FUNCTION_BLOCK Controller

VAR_OUTPUT
	
END_VAR

VAR	
	// 輸入指令，顯示狀態、位置、角度
	command : E_6Axis_Command;	
	state : ST_6Axis_State;
	constructState : UINT;
	touchingState : UINT;
	takeState : UINT;
	JointDegNow : ARRAY [AXIS_MIN_IDX..AXIS_MAX_IDX] OF LREAL;
	PositionNow : ARRAY [AXIS_MIN_IDX..AXIS_MAX_IDX] OF LREAL;
	hasFromCAM : BOOL;
	//StartPosition_Now : ARRAY [AXIS_MIN_IDX..AXIS_MAX_IDX] OF LREAL; // for linear move used
	
	// 開發者使用
	HomePoint : ARRAY [AXIS_MIN_IDX..AXIS_MAX_IDX] OF LREAL := [565, 0, 834, 0, 0, 0];
	HomeJoint : ARRAY [AXIS_MIN_IDX..AXIS_MAX_IDX] OF LREAL := [0, 0, 0, 0, 0, 0]; // for joints space	

	//BufferMot : Motion_Command_Input; // 
	InitalPOS : ARRAY [AXIS_MIN_IDX..AXIS_MAX_IDX] OF LREAL := InitalPOS;
	ActExecute : BOOL := FALSE;
	ExecutePMD : BOOL := FALSE;
	ExecuteCAL : BOOL := FALSE; // 執行一次性計算
 	DIR : LREAL := 0; // XYZ_Direcation XYZ軸方向 = {1:x, 2:y, 3:z, 4:xy, 5:-(xy)}
	PMD : LREAL := 0; // Path_Motion_Displace 路徑移動距離
	TouchDetection : BOOL;
	ZeroArray : ARRAY [AXIS_MIN_IDX..AXIS_MAX_IDX] OF LREAL := [0, 0, 0, 0, 0, 0]; 
	TargetPOS : ARRAY [AXIS_MIN_IDX..AXIS_MAX_IDX] OF LREAL := [650, -150, 500, -42, 0, 45];
	POS_STORAGE : Buffer;

	// 索引
	idx : USINT(AXIS_MIN_IDX..AXIS_MAX_IDX);
	movableBlock_idx : INT;
	i, j : USINT(AXIS_MIN_IDX..AXIS_MAX_IDX);
	z : INT;
	n : ARRAY [1..6] OF LREAL := AutoMotionData.CAMStore[1][0] ;
	usingMotion : INT;
	row, col : INT;
	//ok
	//p : ARRAY [1..2] OF LREAL := AutoMotionData.CAMStore;
	//L : ARRAY [AXIS_MIN_IDX..AXIS_MAX_IDX] OF LREAL ;
	h : INT;
	

	// 基本需要的函式
	Axis : ARRAY[AXIS_MIN_IDX..AXIS_MAX_IDX] OF AXIS_REF;
	Power : ARRAY [AXIS_MIN_IDX..AXIS_MAX_IDX] OF MC_Power;
	Stop : ARRAY [AXIS_MIN_IDX..AXIS_MAX_IDX] OF MC_Stop; //delete
	Halt : ARRAY [AXIS_MIN_IDX..AXIS_MAX_IDX] OF MC_Halt; 
	Reset : ARRAY [AXIS_MIN_IDX..AXIS_MAX_IDX] OF MC_Reset;
	
	// 自訂義函式
	KM : Kinematics;
	MF : MathFunc;
	
	// 移動用函式
	AbsMove : ARRAY [AXIS_MIN_IDX..AXIS_MAX_IDX] OF MC_MoveAbsolute;
	ExtSwitchEn : ARRAY [AXIS_MIN_IDX..AXIS_MAX_IDX] OF MC_ExtSetPointGenEnable;
	ExtSwitchDis : ARRAY [AXIS_MIN_IDX..AXIS_MAX_IDX] OF MC_ExtSetPointGenDisable;
	LinearMove : MC_Linear; 

	// For Curve                         A1  A2  A3  A4  A5  A6
	StartVEL : ARRAY [1..6] OF LREAL := [  0,  0,  0,  0,  0,  0];
	StartACC : ARRAY [1..6] OF LREAL := [  0,  0,  0,  0,  0,  0];
	FinalVEL : ARRAY [1..6] OF LREAL := [  0,  0,  0,  0,  0,  0];
	FinalACC : ARRAY [1..6] OF LREAL := [  0,  0,  0,  0,  0,  0];

	E_Command: INT;
	No_Command: INT;
	PT: TIME;
END_VAR

readAxis();
SetStartPosition();

CASE command OF
	E_6Axis_Command.NO_COMMAND:
		FOR idx := AXIS_MIN_IDX TO AXIS_MAX_IDX DO
			AbsMove[idx].Execute := FALSE;
		END_FOR
		isHalt := FALSE;
		ExecutePMD := FALSE;
		constructState := 0;
		ActExecute := FALSE;
		
	E_6Axis_Command.POWER_ON:
		FOR idx := AXIS_MIN_IDX TO AXIS_MAX_IDX DO
			Power[idx].Enable := TRUE;
		END_FOR
		IF state.powerOn THEN
			command := E_6Axis_Command.HOMING;
		END_IF
	
	E_6Axis_Command.HALT:
		FOR idx := AXIS_MIN_IDX TO AXIS_MAX_IDX DO
			Halt[idx].Execute := TRUE;
		END_FOR
		IF NOT state.moving THEN
			FOR idx := AXIS_MIN_IDX TO AXIS_MAX_IDX DO
				Halt[idx].Execute := FALSE;
			END_FOR
		END_IF
		command := E_6axis_Command.NO_COMMAND;
	
	E_6Axis_Command.RESET:
		FOR idx := AXIS_MIN_IDX TO AXIS_MAX_IDX DO
			Reset[idx].Execute := TRUE;
			IF Reset[idx].Done THEN
				Reset[idx].Execute := FALSE;
			END_IF
		END_FOR
		command := E_6axis_Command.NO_COMMAND;

	// SetMotion(路徑模式，起點，終點，FALSE);		
	E_6Axis_Command.HOMING:
		ActExecute := TRUE;
		SetMotion(0, InitalPOS, HomeJoint, FALSE, TRUE);
		IF NOT ActExecute THEN
			command := E_6axis_Command.NO_COMMAND;
		END_IF

	E_6Axis_Command.M_PTP:
		ActExecute := TRUE;
		SetMotion(0, InitalPOS, TargetPOS, FALSE, FALSE);
		IF NOT ActExecute THEN
			command := E_6axis_Command.NO_COMMAND;
		END_IF
		
	E_6Axis_Command.M_DIRE_X:
		IF NOT ExecutePMD THEN
			MF.VectorMotionPOS(POS := TargetPOS, DIR, PMD);
			ExecutePMD := TRUE;
		END_IF
		ActExecute := TRUE;
		SetMotion(1, InitalPOS, TargetPOS, FALSE, FALSE);
		IF NOT ActExecute THEN
			command := E_6axis_Command.NO_COMMAND;
		END_IF
		
	E_6Axis_Command.M_DIRE_Y:
		IF NOT ExecutePMD THEN
			MF.VectorMotionPOS(POS := TargetPOS, DIR, PMD);
			ExecutePMD := TRUE;
		END_IF
		ActExecute := TRUE;
		SetMotion(1, InitalPOS, TargetPOS, FALSE, FALSE);
		IF NOT ActExecute THEN
			command := E_6axis_Command.NO_COMMAND;
		END_IF
	
	E_6Axis_Command.M_DIRE_XY:
		IF NOT ExecutePMD THEN
			MF.VectorMotionPOS(POS := TargetPOS, DIR, PMD);
			ExecutePMD := TRUE;
		END_IF
		ActExecute := TRUE;
		SetMotion(1, InitalPOS, TargetPOS, FALSE, FALSE);
		IF NOT ActExecute THEN
			command := E_6axis_Command.NO_COMMAND;
		END_IF
		
	E_6Axis_Command.M_DIRE_Z:
		IF NOT ExecutePMD THEN
			MF.VectorMotionPOS(POS := TargetPOS, DIR, PMD);
			ExecutePMD := TRUE;
		END_IF
		ActExecute := TRUE;
		SetMotion(1, InitalPOS, TargetPOS, FALSE, FALSE);
		IF NOT ActExecute THEN
			command := E_6axis_Command.NO_COMMAND;
		END_IF
		
	E_6Axis_Command.M_LINEAR:
		ActExecute := TRUE;
		SetMotion(1, InitalPOS, TargetPOS, FALSE, FALSE);
		IF NOT ActExecute THEN
			command := E_6axis_Command.NO_COMMAND;
		END_IF
		
	E_6Axis_Command.M_CURVE:
		ActExecute := TRUE;
		SetMotion(2, InitalPOS, TargetPOS, FALSE, FALSE);
		IF NOT ActExecute THEN
			command := E_6axis_Command.NO_COMMAND;
		END_IF
		
	E_6Axis_Command.TOUCHING://判斷式
		IF NOT ActExecute THEN
			CASE touchingState OF
				0: //要再加一個判斷式判斷是哪一個位置
					//z := z + 1;            // 疊疊樂右面與左面
					usingMotion := 2;
					
					IF z = 1 THEN
						TargetPOS[1]:= n[1];
						TargetPOS[2]:= n[2];
						TargetPOS[3]:= 500;
						TargetPOS[4]:= 0;
						TargetPOS[5]:= 90;
						TargetPOS[6]:= -45;
					ELSIF z = 2 THEN
						TargetPOS[1]:= n[1];
						TargetPOS[2]:= n[2];
						TargetPOS[3]:= 500;
						TargetPOS[4]:= 0;
						TargetPOS[5]:= 90;
						TargetPOS[6]:= -135;
					END_IF
					      // 移動模式
					//TargetPOS := AutoMotionData.CAMStore[n][z];  // n=0
					//n := n + 1;
					touchingState := touchingState + 1;
				1:
					usingMotion := 1;
					IF z = 1 THEN
						MF.VectorMotionPOS(POS := TargetPOS, 5, -25);
					ELSIF z = 2 THEN
						MF.VectorMotionPOS(POS := TargetPOS, 4, 25);
					END_IF
					//AutoMotionData.POStore[z][n] := TargetPOS;
					//n := n + 1;
					touchingState := touchingState + 1;
				2: 
					usingMotion := 1;
					IF z = 1 THEN
						MF.VectorMotionPOS(POS := TargetPOS, 3, -(500-n[3]));
					ELSIF z = 2 THEN
						MF.VectorMotionPOS(POS := TargetPOS, 3, -(500-n[3]));
					END_IF
					touchingState := touchingState + 1;
				3:
					PT := T#1S;
					input_dig[1] := TRUE;
					PT := T#1S;
					//加計時器
					input_dig[1] := FALSE;
				4:
					usingMotion := 1;
					IF z = 1 THEN
						MF.VectorMotionPOS(POS := TargetPOS, 3, (500-n[3]));
					ELSIF z = 2 THEN
						MF.VectorMotionPOS(POS := TargetPOS, 3, (500-n[3]));
					END_IF
					touchingState := touchingState + 1;
				
				5:
					command := E_6axis_Command.HOMING;
					touchingState := touchingState + 1;
				6:
					command := E_6axis_Command.TAKING;
			END_CASE			
		END_IF
	SetMotion(usingMotion, InitalPOS, TargetPOS, FALSE, FALSE);
	
	E_6Axis_Command.TAKING:
		IF NOT ActExecute THEN
			CASE takeState OF
				0:
					usingMotion := 1;
					input_dig[2] := FALSE;
					
					IF z = 1 THEN
						MF.VectorMotionPOS(POS := TargetPOS, 5, (n[1]+100));
						MF.VectorMotionPOS(POS := TargetPOS, 5, (n[2]+100));
						TargetPOS[3] := 500;
						TargetPOS[4] := 0;
						TargetPOS[5] := -90;
						TargetPOS[6] := 45;
					ELSIF z = 2 THEN
						MF.VectorMotionPOS(POS := TargetPOS, 4, (n[1]-100));
						MF.VectorMotionPOS(POS := TargetPOS, 4, (n[2]-100));
						TargetPOS[3] := 500;
						TargetPOS[4] := 0;
						TargetPOS[5] := -90;
						TargetPOS[6] := -135;
						
					END_IF
					touchingState := touchingState + 1;	
				1:
					usingMotion := 1;
					IF z = 1 THEN
						MF.VectorMotionPOS(POS := TargetPOS, 3, -(500-n[3]));
					ELSIF z = 2 THEN
						MF.VectorMotionPOS(POS := TargetPOS, 3, -(500-n[3]));
					END_IF
					//AutoMotionData.POStore[z][n] := hasFromCAM;
					//n := n + 1;
					touchingState := touchingState + 1;
				2:
					usingMotion := 1; 
					input_dig[2]:= TRUE ;
					PT := T#1S;
					touchingState := touchingState + 1;
				3:
					usingMotion := 1; 
					IF z = 1 THEN
						MF.VectorMotionPOS(POS := TargetPOS, 5, 30);
					ELSIF z = 2 THEN
						MF.VectorMotionPOS(POS := TargetPOS, 4, -30);
					END_IF
					touchingState := touchingState + 1;
				4:
					usingMotion := 1;
					
					MF.VectorMotionPOS(POS := TargetPOS, 3, (AutoMotionData.Heightstore[1]-n[3]+2));
					touchingState := touchingState + 1;
				5:
				   IF z = 1 THEN
						MF.VectorMotionPOS(POS := TargetPOS, 5, -60);
					ELSIF z = 2 THEN
						MF.VectorMotionPOS(POS := TargetPOS, 4, 60);
					END_IF
					PT := T#1S;
					input_dig[2]:= FALSE ;
					touchingState := touchingState + 1;
				6:
					command := E_6axis_Command.HOMING;
					
			END_CASE
		END_IF
		SetMotion(usingMotion, InitalPOS, TargetPOS, FALSE, FALSE);
		ActExecute := TRUE;
				
				
//	E_6Axis_Command.LOOKING:
//		SetMotion(0, InitalPOS, TargetPOS, FALSE);

END_CASE

Decider();
Update_AbsMove_Motion();
Update_Custom_Motion();
ActPower();
ActReset();
ActStop();

//	E_6Axis_Command.CONSTRUCT:
//		IF NOT ActExecute THEN
//			CASE constructState OF
//				0:
//					z := z + 1;            // 疊疊樂右面與左面
//					usingMotion := 2;      // 移動模式
//					TargetPOS := AutoMotionData.POStore[z][n];  // n=0
//					n := n + 1;
//					constructState := constructState + 1;
//				1:
//					usingMotion := 1;
//					IF z = 1 THEN
//						MF.VectorMotionPOS(POS := TargetPOS, 4, 90);
//					ELSIF z = 2 THEN
//						MF.VectorMotionPOS(POS := TargetPOS, 5, 90);
//					END_IF
//					AutoMotionData.POStore[z][n] := TargetPOS;
//					n := n + 1;
//					constructState := constructState + 1;
//				2:
//					usingMotion := 1;
//					IF z = 1 THEN
//						MF.VectorMotionPOS(POS := TargetPOS, 3, -95);
//					ELSIF z = 2 THEN
//						MF.VectorMotionPOS(POS := TargetPOS, 3, -110);
//					END_IF					
//					AutoMotionData.POStore[z][n] := TargetPOS;
//					n := n + 1;
//					constructState := constructState + 1;
//				3:
//					usingMotion := 1;
//					TouchDetection := TRUE;
//					ExecuteCAL := FALSE;
//					IF z = 1 THEN
//						MF.VectorMotionPOS(POS := TargetPOS, 4, -40);
//					ELSIF z = 2 THEN
//						MF.VectorMotionPOS(POS := TargetPOS, 5, -40);
//					END_IF	
//					AutoMotionData.POStore[z][n] := TargetPOS;
//					n := n + 1;
//					movableBlock_idx := movableBlock_idx + 1;
//					constructState := constructState + 1;
//				4:
//					usingMotion := 1;
//					TouchDetection := FALSE;
//					row := row + 1;
//					IF z = 1 THEN
//						MF.VectorMotionPOS(POS := TargetPOS, 4, 40);
//					ELSIF z = 2 THEN
//						MF.VectorMotionPOS(POS := TargetPOS, 5, 40);
//					END_IF	
//					AutoMotionData.POStore[z][n] := TargetPOS;
//					n := n + 1; 
//					constructState := constructState + 1;
//					IF row = 3 THEN
//						row := 0;
//						constructState := 6;
//						col := col + 1;
//						IF col = 4 THEN
//							constructState := 8;
//						END_IF
//					END_IF
//				5:
//					usingMotion := 1;
//					IF z = 1 THEN
//						MF.VectorMotionPOS(POS := TargetPOS, 5, -25);
//					ELSIF z = 2 THEN
//						MF.VectorMotionPOS(POS := TargetPOS, 4, -25);
//					END_IF	
//					AutoMotionData.POStore[z][n] := TargetPOS;
//					n := n + 1;
//					constructState := 3;
//				6:
//					usingMotion := 1;
//					MF.VectorMotionPOS(POS := TargetPOS, 3, -30);
//					AutoMotionData.POStore[z][n] := TargetPOS;
//					n := n + 1;
//					constructState := constructState + 1;
//				7:
//					usingMotion := 1;
//					IF z = 1 THEN
//						MF.VectorMotionPOS(POS := TargetPOS, 5, 50);
//					ELSIF z = 2 THEN
//						MF.VectorMotionPOS(POS := TargetPOS, 4, 50);
//					END_IF	
//					AutoMotionData.POStore[z][n] := TargetPOS;
//					n := n + 1;
//					constructState := 3;
//				8:
//					usingMotion := 2;
//					TargetPOS := AutoMotionData.POStore[z][1];
//					constructState := 9;
//				9:
//					usingMotion := 2;
//					TargetPOS := HomePoint;
//					n := 0;
//					row := 0;
//					col := 0;
//					constructState := 0;
//					IF z = 2 THEN
//						constructState := 10;
//					END_IF
//				10:
//					command := E_6axis_Command.HOMING;
//					constructState := 11;
//			END_CASE
//		END_IF
//		ActExecute := TRUE;
//		IF TouchDetection THEN
//			IF input_dig[1] THEN
//				IF NOT ExecuteCAL THEN
//					AutoMotionData.MovableBlocks[movableBlock_idx] := ZeroArray;
//					movableBlock_idx := movableBlock_idx - 1;
//					ExecuteCAL := TRUE;
//				END_IF
//			ELSE
//				// 減2是為了擷取上一個座標
//				AutoMotionData.MovableBlocks[movableBlock_idx] := AutoMotionData.POStore[z][n-2];
//			END_IF
//		END_IF

//		IF NOT (constructState = 11) THEN
//			SetMotion(usingMotion, InitalPOS, TargetPOS, FALSE, FALSE);
//		ELSE
//			z := 0;
//		END_IF

ACTION ActHalt:
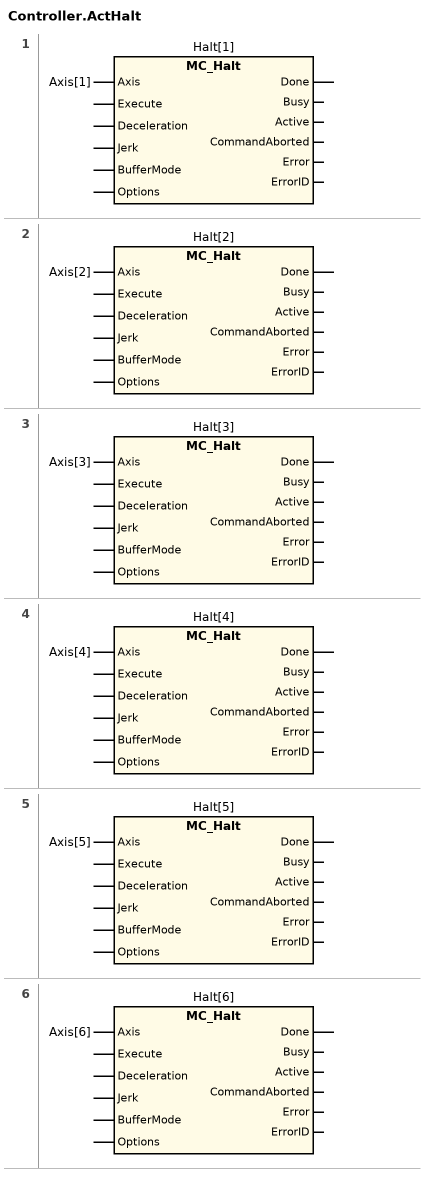
// NETWORK 1
Halt[1](Axis := Axis[1]); // MC_Halt

// NETWORK 2
Halt[2](Axis := Axis[2]); // MC_Halt

// NETWORK 3
Halt[3](Axis := Axis[3]); // MC_Halt

// NETWORK 4
Halt[4](Axis := Axis[4]); // MC_Halt

// NETWORK 5
Halt[5](Axis := Axis[5]); // MC_Halt

// NETWORK 6
Halt[6](Axis := Axis[6]); // MC_Halt
END_ACTION

ACTION ActPower:
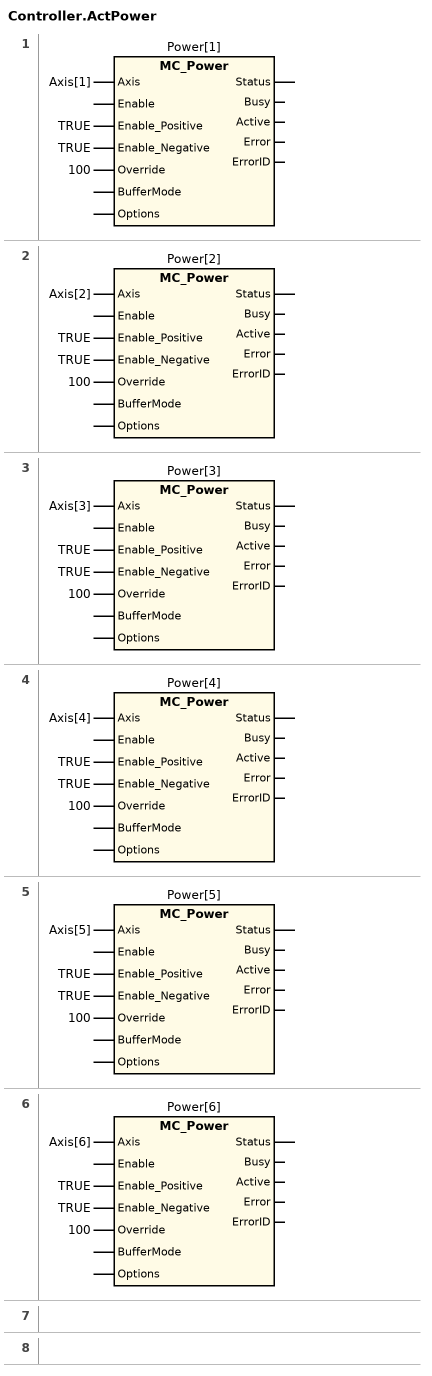
// NETWORK 1
Power[1](Axis := Axis[1], Enable_Positive := TRUE, Enable_Negative := TRUE, Override := 100); // MC_Power

// NETWORK 2
Power[2](Axis := Axis[2], Enable_Positive := TRUE, Enable_Negative := TRUE, Override := 100); // MC_Power

// NETWORK 3
Power[3](Axis := Axis[3], Enable_Positive := TRUE, Enable_Negative := TRUE, Override := 100); // MC_Power

// NETWORK 4
Power[4](Axis := Axis[4], Enable_Positive := TRUE, Enable_Negative := TRUE, Override := 100); // MC_Power

// NETWORK 5
Power[5](Axis := Axis[5], Enable_Positive := TRUE, Enable_Negative := TRUE, Override := 100); // MC_Power

// NETWORK 6
Power[6](Axis := Axis[6], Enable_Positive := TRUE, Enable_Negative := TRUE, Override := 100); // MC_Power

// NETWORK 7

// NETWORK 8
END_ACTION

ACTION ActReset:
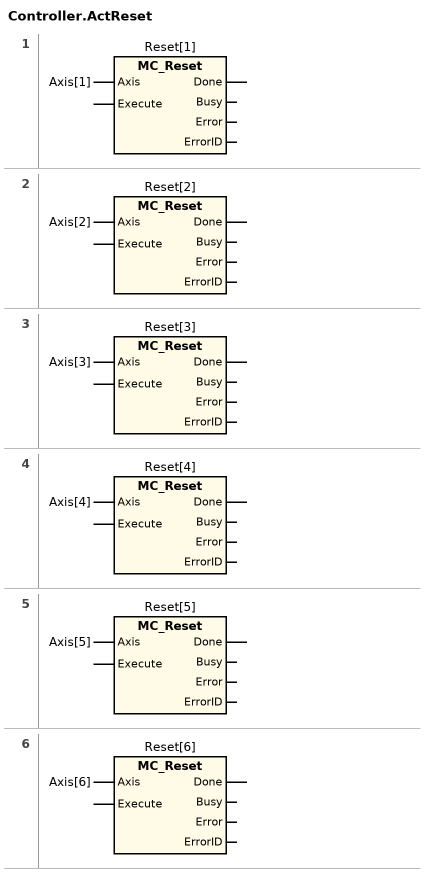
// NETWORK 1
Reset[1](Axis := Axis[1]); // MC_Reset

// NETWORK 2
Reset[2](Axis := Axis[2]); // MC_Reset

// NETWORK 3
Reset[3](Axis := Axis[3]); // MC_Reset

// NETWORK 4
Reset[4](Axis := Axis[4]); // MC_Reset

// NETWORK 5
Reset[5](Axis := Axis[5]); // MC_Reset

// NETWORK 6
Reset[6](Axis := Axis[6]); // MC_Reset
END_ACTION

ACTION ActStop:
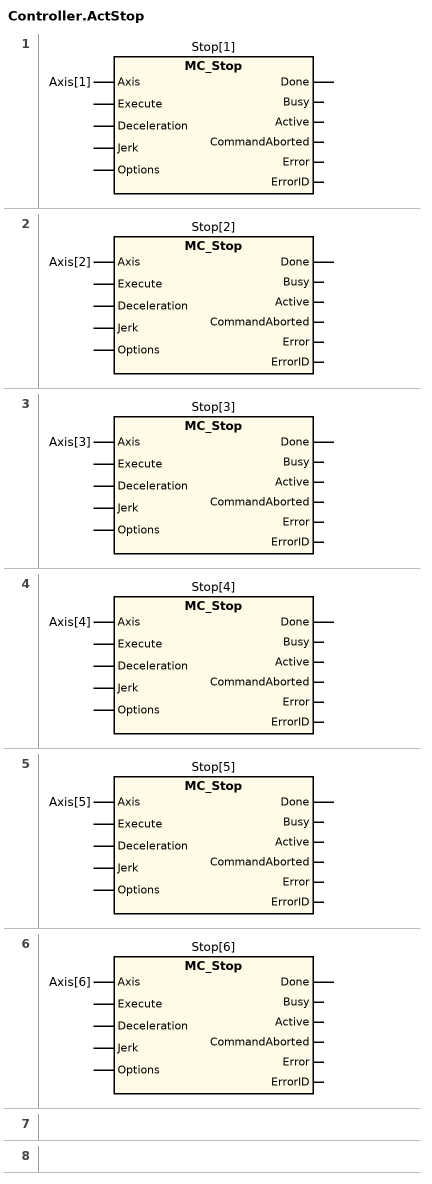
// NETWORK 1
Stop[1](Axis := Axis[1]); // MC_Stop

// NETWORK 2
Stop[2](Axis := Axis[2]); // MC_Stop

// NETWORK 3
Stop[3](Axis := Axis[3]); // MC_Stop

// NETWORK 4
Stop[4](Axis := Axis[4]); // MC_Stop

// NETWORK 5
Stop[5](Axis := Axis[5]); // MC_Stop

// NETWORK 6
Stop[6](Axis := Axis[6]); // MC_Stop

// NETWORK 7

// NETWORK 8
END_ACTION

ACTION Decider:
IF NOT state.moving AND AbsMove[1].Done AND AbsMove[2].Done AND AbsMove[3].Done AND AbsMove[4].Done  AND AbsMove[5].Done AND AbsMove[6].Done THEN
	command := E_6axis_Command.NO_COMMAND;	
END_IF

IF state.error THEN
	command := E_6Axis_Command.RESET;
END_IF

IF isHalt THEN
	command := E_6Axis_Command.HALT;
END_IF
END_ACTION

METHOD mode_Curve : BOOL

VAR_INPUT
	six_mat : ARRAY [1..6, 1..6] OF LREAL;
END_VAR

VAR_OUTPUT
	execute_fullTime : LREAL;
	coeffCopy : ARRAY [1..6, 1..6] OF LREAL;
END_VAR

VAR
	idx : DINT;
	i, j : INT;
	t : LREAL;
	temp : LREAL; // 導正係數用
	
	startAngles : ARRAY [1..6] OF LREAL;
	finalAngles : ARRAY [1..6] OF LREAL;
	pos01, pos02 : ARRAY [1..3] OF LREAL; //start and final point for calculate fulltime
	
	six_matCopy : ARRAY [1..6, 1..6] OF LREAL;
	TimeMatrix : ARRAY [1..6, 1..6] OF LREAL;
END_VAR
// Angles_mat
six_matCopy := six_mat;  // 含有角度 := 含有座標
FOR idx := 1 TO 6 DO 
	IF (idx < 3) THEN
		pos01[idx] := six_mat[idx, 1];
		pos02[idx] := six_mat[idx, 4];
	END_IF
	startAngles[idx] := six_mat[idx, 1];
	finalAngles[idx] := six_mat[idx, 4];
END_FOR
KM.Inverse(position := startAngles, degrees => startAngles);
KM.Inverse(position := finalAngles, degrees => finalAngles);
FOR idx := 1 TO 6 DO 
	six_matCopy[idx, 1] := startAngles[idx];
	six_matCopy[idx, 4] := finalAngles[idx];
END_FOR

MF.FindFullTime(pos01, pos02, 10, execute_fullTime => execute_fullTime);
t := execute_fullTime;
// Time_mat
FOR i := 1 TO 6 DO
    FOR j := 1 TO 6 DO
        CASE j OF
            1: 
                // 第一列固定為1、0、0、0、0、0
                TimeMatrix[i, j] := SEL(i = 1, 0, 1);
            2: 
                // 第二列固定為0、1、0、0、0、0
                TimeMatrix[i, j] := SEL(i = 2, 0, 1);
            3:
                // 第三列固定為0、0、2、0、0、0
                TimeMatrix[i, j] := SEL(i = 3, 0, 2);
            4:
                // 第四列公式：1 * EXPT(t, i)
                TimeMatrix[i, j] := EXPT(t, i-1);
            5:
                // 第五列公式：i * EXPT(t, i-1)
                TimeMatrix[i, j] := (i-1) * EXPT(t, i-2);
            6:
                // 第六列公式：(i * (i - 1)) * EXPT(t, i-2)
                TimeMatrix[i, j] := (i-1) * (i-2) * EXPT(t, i-3);
        END_CASE
    END_FOR
END_FOR

MF.GaussianElimination(base_mat := TimeMatrix, extend_mat := six_matCopy, temp_mat := coeffCopy, 6); //inverse 會搞壞原本的東西

FOR i := 1 TO 6 DO
	FOR j := 1 TO 3 DO
		temp := coeffCopy[i, j];
		coeffCopy[i, j] := coeffCopy[i, 7-j];
		coeffCopy[i, 7-j] := temp;
	END_FOR		
END_FOR
END_METHOD

METHOD mode_Linear : BOOL

VAR_INPUT
	six_pos : ARRAY [1..6, 1..6] OF LREAL;
END_VAR

VAR_OUTPUT
	execute_fullTime : LREAL;
	coeffCopy : ARRAY [1..6, 1..6] OF LREAL;
END_VAR

VAR
	idx : DINT;
	i, j : DINT;
	temp : LREAL; // 導正係數用

	pos01, pos02 : ARRAY [1..3] OF LREAL; //start and final point
	temp_pos : ARRAY [1..6] OF LREAL;
	temp_ang : ARRAY [1..6] OF LREAL;
	six_pos_angles : ARRAY [1..6, 1..6] OF LREAL;
	
	six_time : ARRAY [1..6, 1..6] OF LREAL;
	timeCopy : ARRAY [1..6, 1..6] OF LREAL;
	
END_VAR
// Angles_mat
FOR i := 1 TO 6 DO
	FOR j := 1 TO 6 DO
		temp_pos[j] := six_pos[i, j];
	END_FOR
	KM.Inverse(position := temp_pos, degrees => temp_ang);
	FOR j := 1 TO 6 DO
		six_pos_angles[j, i] := temp_ang[j];
	END_FOR
END_FOR

FOR idx := 1 TO 3 DO 
	pos01[idx] := six_pos[1, idx];
	pos02[idx] := six_pos[6, idx];
END_FOR
MF.FindFullTime(pos01, pos02, 10, execute_fullTime => execute_fullTime);

// Time_mat
FOR i := 1 TO 6 DO
	six_time[1, i] := 1;
	six_time[2, i] := (execute_fullTime)/5 * (i-1);
	FOR j := 3 TO 6 DO
		six_time[j, i] := EXPT(six_time[2, i], j-1);
	END_FOR
END_FOR

FOR i := 1 TO 6 DO
	FOR j := 1 TO 6 DO
		coeffCopy[i, j] := 0; // clear temp
		timeCopy[i, j] := six_time[i, j];
	END_FOR
END_FOR

MF.GaussianElimination(base_mat := timeCopy, extend_mat := six_pos_angles, temp_mat := coeffCopy, 6); //inverse 會搞壞原本的東西

FOR i := 1 TO 6 DO
	FOR j := 1 TO 3 DO
		temp := coeffCopy[i, j];
		coeffCopy[i, j] := coeffCopy[i, 7-j];
		coeffCopy[i, 7-j] := temp;
	END_FOR		
END_FOR
END_METHOD

METHOD mode_PTP : BOOL

VAR_INPUT
	angles01 : ARRAY [1..6] OF LREAL; // start position (degree)
	angles02 : ARRAY [1..6] OF LREAL; // final position (degree)
END_VAR

VAR
	idx : DINT;
	
	longest_distance : LREAL := 0;
	//time_factor : LREAL;
	execute_fullTime : LREAL := 3;
	
END_VAR
//// Execute Time
//FOR idx := 1 TO 6 DO
//	longest_distance := MAX(longest_distance, ABS(angles02[idx] - angles01[idx]));
//END_FOR
//time_factor := EXPT(30, -1); // The larger the denominator, the faster the speed
//execute_fullTime := time_factor * longest_distance;
//execute_fullTime := LREAL_TO_DINT(execute_fullTime * 1000)/1000; // Adjust Time
//IF execute_fullTime < 0.01 THEN
//	execute_fullTime := 3;
//END_IF

FOR idx := 1 TO 6 DO
	AbsMove[idx].Position := angles02[idx];
	AbsMove[idx].Velocity := ABS(angles02[idx] - Axis[idx].NcToPlc.ActPos) / execute_fullTime;
	IF AbsMove[Idx].Velocity < 0.001 THEN
		AbsMove[Idx].Velocity := 0.001;  // Module Minium Limit
	END_IF
END_FOR
END_METHOD

METHOD readAxis : BOOL

VAR
	
END_VAR
FOR idx := AXIS_MIN_IDX TO AXIS_MAX_IDX DO
	Axis[idx]();
	JointDegNow[idx] := Axis[idx].NcToPlc.ActPos;
END_FOR
KM.Forward(angles := JointDegNow, position => PositionNow);

state.powerOn := Power[1].Status AND Power[2].Status AND Power[3].Status AND Power[4].Status AND Power[5].Status AND Power[6].Status;
state.stop := Stop[1].Done AND Stop[2].Done AND Stop[3].Done AND Stop[4].Done AND Stop[5].Done AND Stop[6].Done;
state.moving := Axis[1].Status.Moving OR Axis[2].Status.Moving OR Axis[3].Status.Moving OR  Axis[4].Status.Moving OR Axis[5].Status.Moving OR Axis[6].Status.Moving;
//state.pause := NOT (state.moving OR state.stop);
state.error := Axis[1].Status.Error OR Axis[2].Status.Error OR Axis[3].Status.Error OR Axis[4].Status.Error OR Axis[5].Status.Error OR Axis[6].Status.Error;
END_METHOD

METHOD SetMotion : BOOL

VAR_INPUT
	mode : DINT;
	StartPOS : ARRAY [1..6] OF LREAL;
	FinalPOS : ARRAY [1..6] OF LREAL;
	isSIM : BOOL;
	precise : BOOL; // 專門給Homing指令使用
	
END_VAR

VAR_OUTPUT
	runTime : LREAL;
	coeffCopy : ARRAY[1..6, 1..6] OF LREAL;
END_VAR

VAR
	// PTP
	ptpAngles_01 : ARRAY [1..6] OF LREAL;
	ptpAngles_02 : ARRAY [1..6] OF LREAL;
	
	// Linear
	six_pos : ARRAY [1..6, 1..6] OF LREAL;

	
	// Curve 
	six_mat : ARRAY [1..6, 1..6] OF LREAL;
	
	// Linear & Curve
	customAngles : ARRAY [1..6] OF LREAL;  // deg & rad

	PTPMove_done : BOOL;
END_VAR


CASE mode OF
	0: // PTP
		FOR idx := AXIS_MIN_IDX TO AXIS_MAX_IDX DO
			AbsMove[idx].Execute := TRUE;
			IF NOT precise THEN
				KM.Inverse(position := StartPOS, degrees => ptpAngles_01);
				KM.Inverse(position := FinalPOS, degrees => ptpAngles_02);
				mode_PTP(ptpAngles_01, ptpAngles_02);
			ELSE
				AbsMove[idx].Position := HomeJoint[idx];
				AbsMove[idx].Velocity := 5;
			END_IF
		END_FOR		
		
		PTPMove_done := TRUE;
		FOR idx := 1 TO 6 DO
			IF NOT AbsMove[idx].Done THEN
				PTPMove_done := FALSE;
				EXIT;
			END_IF
		END_FOR
		
	1: // LINEAR
		KM.Inverse(position := FinalPOS, degrees => customAngles);
								
		FOR idx := AXIS_MIN_IDX TO AXIS_MAX_IDX DO
			ExtSwitchEn[idx].Position := customAngles[idx];
			ExtSwitchEn[idx].Execute := TRUE;
			ExtSwitchDis[idx].Execute := FALSE;
		END_FOR
		
		MF.FindForSixPoints(StartPOS, FinalPOS, six_pos => six_pos);
		mode_Linear(six_pos, coeffCopy => coeffCopy, execute_fullTime => runTime);
		
		LinearMove.Execute := TRUE;
		LinearMove.CoeffCopy := coeffCopy;
		LinearMove.RunTime := runTime;
	
	2: // CURVE
		KM.Inverse(position := FinalPOS, degrees => customAngles);
		
		FOR idx := AXIS_MIN_IDX TO AXIS_MAX_IDX DO
			ExtSwitchEn[idx].Position := customAngles[idx];
			ExtSwitchEn[idx].Execute := TRUE;
			ExtSwitchDis[idx].Execute := FALSE;
		END_FOR

		FOR idx := AXIS_MIN_IDX TO AXIS_MAX_IDX DO
			six_mat[idx, 1] :=  StartPOS[idx];
			six_mat[idx, 2] :=  StartVEL[idx];
			six_mat[idx, 3] :=  StartACC[idx];
			six_mat[idx, 4] :=  FinalPOS[idx];
			six_mat[idx, 5] :=  FinalVEL[idx];
			six_mat[idx, 6] :=  FinalACC[idx];
		END_FOR
		mode_Curve(six_mat, coeffCopy => coeffCopy, execute_fullTime => runTime);
		
		LinearMove.Execute := TRUE;
		LinearMove.CoeffCopy := coeffCopy;
		LinearMove.RunTime := runTime;
END_CASE

IF NOT isSIM AND (PTPMove_done OR LinearMove.Done) THEN
	// SetStartPosition
	IF precise THEN
		InitalPOS := HomePoint;
	ELSE

		LinearMove.Execute := FALSE;
		//running := FALSE;
		FOR idx := AXIS_MIN_IDX TO AXIS_MAX_IDX DO
			AbsMove[idx].Execute := FALSE;
			ExtSwitchEn[idx].Execute := FALSE;
			ExtSwitchDis[idx].Execute := TRUE;
		END_FOR
		InitalPOS := FinalPOS;
	END_IF
	ActExecute := FALSE;
END_IF
END_METHOD

ACTION SetStartPosition:
// IDEAL SET STARTPOSISTION
//IF NOT state.moving THEN
//	StartPosition_Now := PositionNow;
//END_IF
END_ACTION

ACTION Update_AbsMove_Motion:
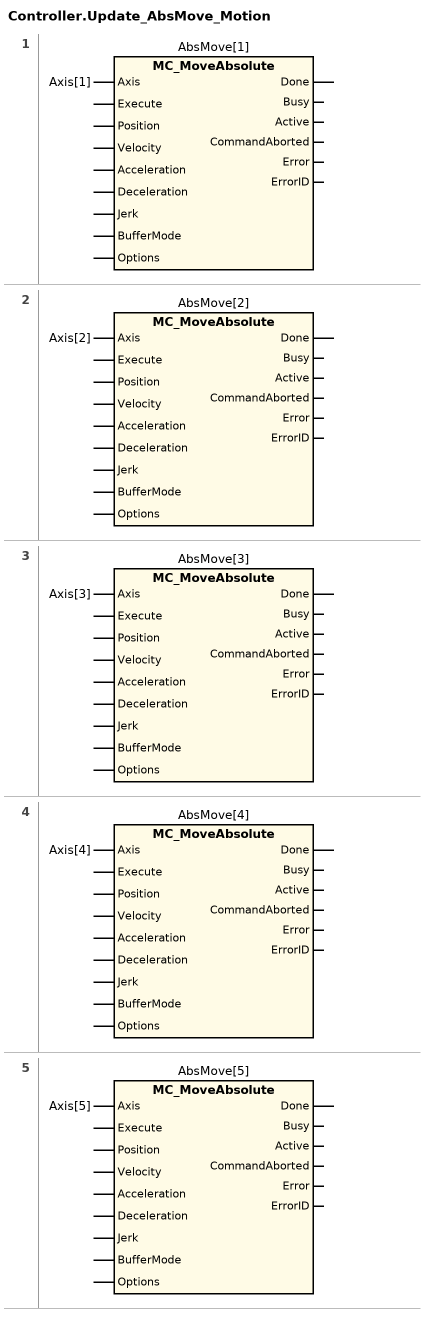
// NETWORK 1
AbsMove[1](Axis := Axis[1]); // MC_MoveAbsolute

// NETWORK 2
AbsMove[2](Axis := Axis[2]); // MC_MoveAbsolute

// NETWORK 3
AbsMove[3](Axis := Axis[3]); // MC_MoveAbsolute

// NETWORK 4
AbsMove[4](Axis := Axis[4]); // MC_MoveAbsolute

// NETWORK 5
AbsMove[5](Axis := Axis[5]); // MC_MoveAbsolute

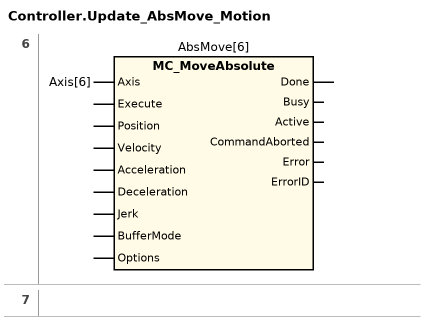
// NETWORK 6
AbsMove[6](Axis := Axis[6]); // MC_MoveAbsolute

// NETWORK 7
END_ACTION

ACTION Update_Custom_Motion:
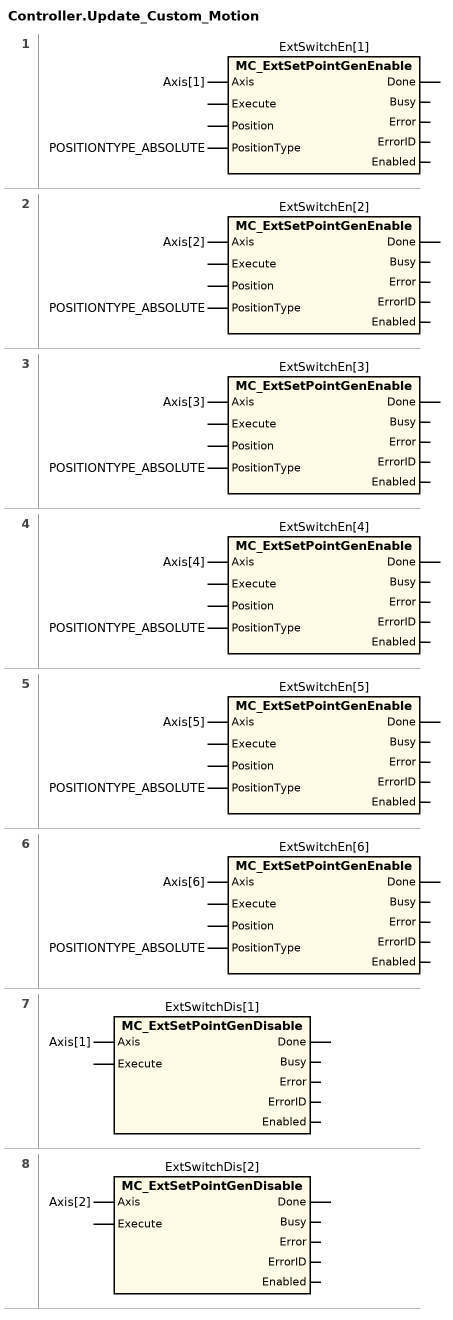
// NETWORK 1
ExtSwitchEn[1](Axis := Axis[1], PositionType := POSITIONTYPE_ABSOLUTE); // MC_ExtSetPointGenEnable

// NETWORK 2
ExtSwitchEn[2](Axis := Axis[2], PositionType := POSITIONTYPE_ABSOLUTE); // MC_ExtSetPointGenEnable

// NETWORK 3
ExtSwitchEn[3](Axis := Axis[3], PositionType := POSITIONTYPE_ABSOLUTE); // MC_ExtSetPointGenEnable

// NETWORK 4
ExtSwitchEn[4](Axis := Axis[4], PositionType := POSITIONTYPE_ABSOLUTE); // MC_ExtSetPointGenEnable

// NETWORK 5
ExtSwitchEn[5](Axis := Axis[5], PositionType := POSITIONTYPE_ABSOLUTE); // MC_ExtSetPointGenEnable

// NETWORK 6
ExtSwitchEn[6](Axis := Axis[6], PositionType := POSITIONTYPE_ABSOLUTE); // MC_ExtSetPointGenEnable

// NETWORK 7
ExtSwitchDis[1](Axis := Axis[1]); // MC_ExtSetPointGenDisable

// NETWORK 8
ExtSwitchDis[2](Axis := Axis[2]); // MC_ExtSetPointGenDisable

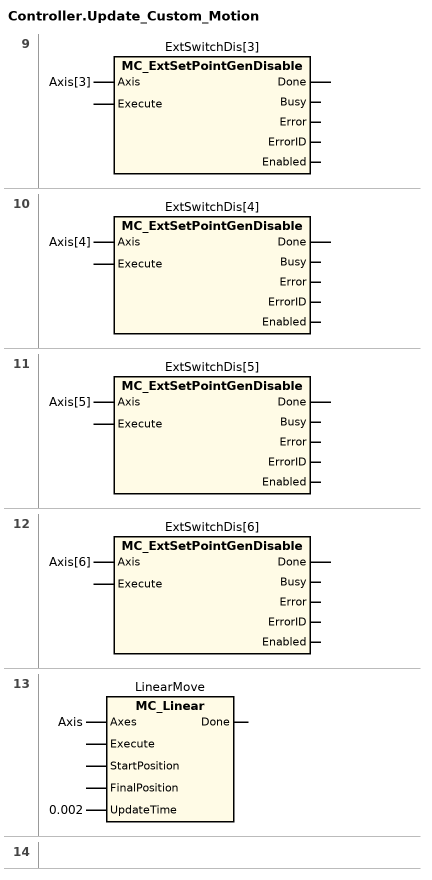
// NETWORK 9
ExtSwitchDis[3](Axis := Axis[3]); // MC_ExtSetPointGenDisable

// NETWORK 10
ExtSwitchDis[4](Axis := Axis[4]); // MC_ExtSetPointGenDisable

// NETWORK 11
ExtSwitchDis[5](Axis := Axis[5]); // MC_ExtSetPointGenDisable

// NETWORK 12
ExtSwitchDis[6](Axis := Axis[6]); // MC_ExtSetPointGenDisable

// NETWORK 13
LinearMove(Axes := Axis, UpdateTime := 0.002); // MC_Linear

// NETWORK 14
END_ACTION

END_FUNCTION_BLOCK

(* stored: Version 1.1.0.1, ProductVersion 3.1.4024.13
   POU Controller: Id {d85eeb7a-7828-4eea-9de8-5b49fe19e8b9}, SpecialFunc None
   Action ActHalt: Id {44558a6f-8ccd-483b-abe6-c588b3eb3d11}
   Action ActPower: Id {c3eeae36-d769-4e1a-aa08-55704f8ad648}
   Action ActReset: Id {0574d424-2545-4ff0-8637-30fc80266883}
   Action ActStop: Id {64d4d7a6-ae28-4a6a-8a4f-bf6b60852155}
   Action Decider: Id {bac3a418-a414-4488-9e33-58addc59d52f}
   Method mode_Curve: Id {381fba53-f73b-4b93-85d9-b889ebfea51f}
   Method mode_Linear: Id {310310d0-39e9-4a3a-9fe5-7de3f5581016}
   Method mode_PTP: Id {07538b52-f2a1-4c76-9f8b-1074df334e7a}
   Method readAxis: Id {ba379574-a876-4daa-b1b9-555b1a112c69}
   Method SetMotion: Id {b6066e64-9dbd-407d-bfe0-070f492f4dbe}
   Action SetStartPosition: Id {b2a07246-ee47-416b-9155-e61bb6cc0759}
   Action Update_AbsMove_Motion: Id {0fa0cb91-03cb-4036-87db-d890a57ebb64}
   Action Update_Custom_Motion: Id {3582fa84-2718-4e34-b3be-b419c476ca0a} *)
